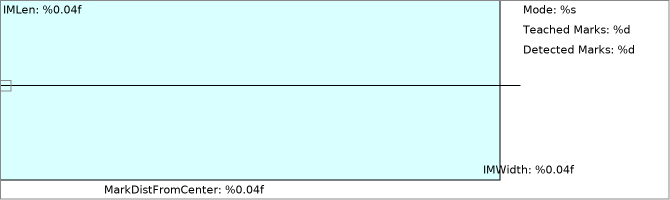
VISUALIZATION _VISU_MarkOverview  // 670x200
VAR_IN_OUT
  mInst : FB_MarkCamera_WEU;
END_VAR
    Rectangle (0,0 500x180)
    Rectangle (0,0 150x20), "IMLen: %0.04f", text variable: mInst._fImageLength
    Rectangle (480,160 150x20), "IMWidth: %0.04f", text variable: mInst._fImageWidth
        p2858320360: -90
    Line (0,85) (520,85)
    Rectangle (101,180 220x20), "MarkDistFromCenter: %0.04f", text variable: mInst.fMarkDistFromCenter
        p2858320360: -90
    Frame (0,80 11x11)
        shows _VISU_MarkViewMini(mInst := mInst.fbMarkDefinition.sMarkDef[1])
    Frame (0,80 11x11)
        shows _VISU_MarkViewMini(mInst := mInst.fbMarkDefinition.sMarkDef[2])
    Frame (0,80 11x11)
        shows _VISU_MarkViewMini(mInst := mInst.fbMarkDefinition.sMarkDef[3])
    Frame (0,80 11x11)
        shows _VISU_MarkViewMini(mInst := mInst.fbMarkDefinition.sMarkDef[4])
    Frame (0,80 11x11)
        shows _VISU_MarkViewMini(mInst := mInst.fbMarkDefinition.sMarkDef[5])
    Frame (0,80 11x11)
        shows _VISU_MarkViewMini(mInst := mInst.fbMarkDefinition.sMarkDef[6])
    Frame (0,80 11x11)
        shows _VISU_MarkViewMini(mInst := mInst.fbMarkDefinition.sMarkDef[7])
    Frame (0,80 11x11)
        shows _VISU_MarkViewMini(mInst := mInst.fbMarkDefinition.sMarkDef[8])
    Frame (0,80 11x11)
        shows _VISU_MarkViewMini(mInst := mInst.fbMarkDefinition.sMarkDef[9])
    Frame (0,80 11x11)
        shows _VISU_MarkViewMini(mInst := mInst.fbMarkDefinition.sMarkDef[10])
    Frame (0,80 11x11)
        shows _VISU_MarkViewMini(mInst := mInst.fbMarkDefinition.sMarkDef[11])
    Frame (0,80 11x11)
        shows _VISU_MarkViewMini(mInst := mInst.fbMarkDefinition.sMarkDef[12])
    Frame (0,80 11x11)
        shows _VISU_MarkViewMini(mInst := mInst.fbMarkDefinition.sMarkDef[13])
    Frame (0,80 11x11)
        shows _VISU_MarkViewMini(mInst := mInst.fbMarkDefinition.sMarkDef[15])
    Frame (0,80 11x11)
        shows _VISU_MarkViewMini(mInst := mInst.fbMarkDefinition.sMarkDef[18])
    Frame (0,80 11x11)
        shows _VISU_MarkViewMini(mInst := mInst.fbMarkDefinition.sMarkDef[16])
    Frame (0,80 11x11)
        shows _VISU_MarkViewMini(mInst := mInst.fbMarkDefinition.sMarkDef[17])
    Frame (0,80 11x11)
        shows _VISU_MarkViewMini(mInst := mInst.fbMarkDefinition.sMarkDef[19])
    Frame (0,80 11x11)
        shows _VISU_MarkViewMini(mInst := mInst.fbMarkDefinition.sMarkDef[20])
    Frame (0,80 11x11)
        shows _VISU_MarkViewMini(mInst := mInst.fbMarkDefinition.sMarkDef[21])
    Frame (0,80 11x11)
        shows _VISU_MarkViewMini(mInst := mInst.fbMarkDefinition.sMarkDef[22])
    Frame (0,80 11x11)
        shows _VISU_MarkViewMini(mInst := mInst.fbMarkDefinition.sMarkDef[23])
    Frame (0,80 11x11)
        shows _VISU_MarkViewMini(mInst := mInst.fbMarkDefinition.sMarkDef[24])
    Frame (0,80 11x11)
        shows _VISU_MarkViewMini(mInst := mInst.fbMarkDefinition.sMarkDef[25])
    Frame (0,80 11x11)
        shows _VISU_MarkViewMini(mInst := mInst.fbMarkDefinition.sMarkDef[26])
    Frame (0,80 11x11)
        shows _VISU_MarkViewMini(mInst := mInst.fbMarkDefinition.sMarkDef[27])
    Frame (0,80 11x11)
        shows _VISU_MarkViewMini(mInst := mInst.fbMarkDefinition.sMarkDef[28])
    Frame (0,80 11x11)
        shows _VISU_MarkViewMini(mInst := mInst.fbMarkDefinition.sMarkDef[29])
    Frame (0,80 11x11)
        shows _VISU_MarkViewMini(mInst := mInst.fbMarkDefinition.sMarkDef[30])
    Rectangle (520,20 150x20), "Teached Marks: %d", text variable: mInst._nTeachedPoints, colour toggle: mInst._bTeachOk
    Rectangle (520,40 150x20), "Detected Marks: %d", text variable: mInst._nDetectedMarks, colour toggle: mInst._nDetectedMarks = mInst._nTeachedPoints AND mInst._nTeachedPoints > 0
    Rectangle (520,0 150x20), "Mode: %s", text variable: mInst.eMarkMode
    Frame (0,80 11x11)
        shows _VISU_MarkViewMini(mInst := mInst.fbMarkDefinition.sMarkDef[14])
END_VISUALIZATION

(* stored: Version 1.1.0.1, ProductVersion 3.1.4024.11
   Visu _VISU_MarkOverview: Id {8e3717a0-37b4-47a7-b7ff-d7a0491ad7b9} *)
